(* PLC project Makefile Example, Unknown Unnamed 1 *)
(* stored: creationDateTime 2014-01-19T11:14:47, contentDescription This example shows how you can customize build process by using 'make'., modificationDateTime 2018-08-24T13:12:10 *)

PROGRAM program0
  VAR
    LocalVara : INT;
    LocalVarb : INT;
  END_VAR

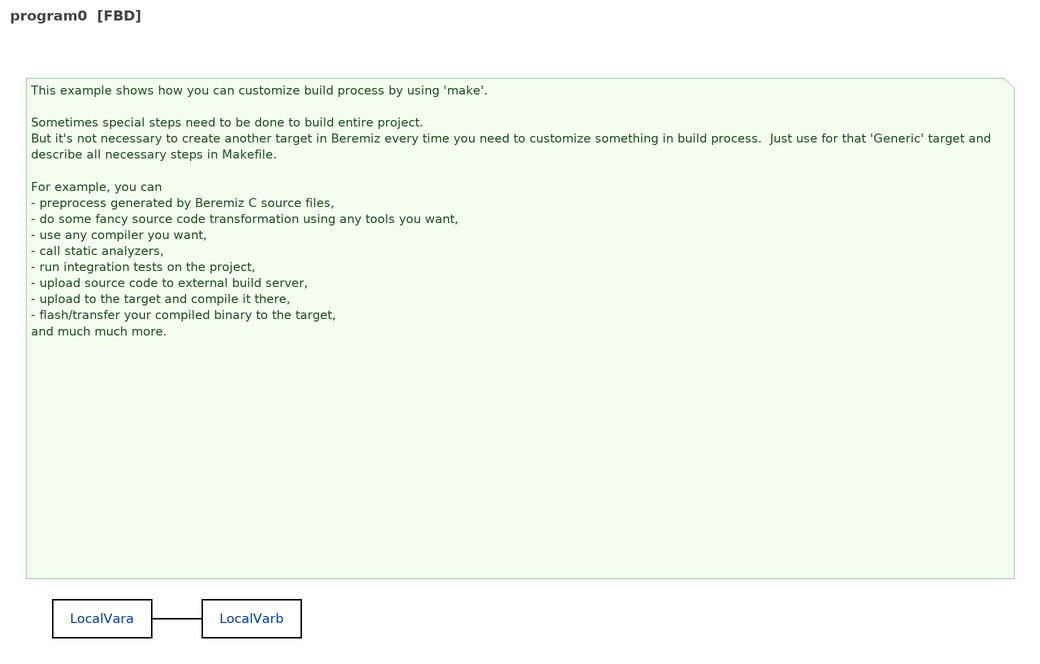
(* FBD diagram, written out as Structured Text *)
(* This example shows how you can customize build process by using 'make'.

Sometimes special steps need to be done to build entire project.
But it's not necessary to create another target in Beremiz every time you need to customize something in build process.  Just use for that 'Generic' target and describe all necessary steps in Makefile. 

For example, you can 
 - preprocess generated by Beremiz C source files, 
 - do some fancy source code transformation using any tools you want, 
 - use any compiler you want,
 - call static analyzers,
 - run integration tests on the project,
 - upload source code to external build server,
 - upload to the target and compile it there,
 - flash/transfer your compiled binary to the target,
 and much much more. *)
LocalVarb := LocalVara;
END_PROGRAM

CONFIGURATION config
  RESOURCE resource1 ON PLC
    TASK Tsk(INTERVAL := T#100ms, PRIORITY := 0);
    PROGRAM Inst WITH Tsk : program0;
  END_RESOURCE
END_CONFIGURATION
